// TIA Portal V17 export
// export: Created 2025-03-05T07:59:12.9568395Z, ExportSetting WithDefaults, DisplayName Totally Integrated Automation Portal, DisplayVersion V17 Update 8, DisplayName TIA Portal Openness, DisplayVersion V17 Update 8, DisplayName TIA Portal Version Control Interface, DisplayVersion V17, DisplayName SINAMICS Startdrive Advanced, DisplayVersion V17 SP2, DisplayName SINAMICS Startdrive G110M, G120, G120C, G120D, G120P, G115D, DisplayVersion V17 SP2, DisplayName SINAMICS Startdrive G130, G150, S120, S150, SINAMICS MV, S210, DisplayVersion V17 SP2, DisplayName STEP 7 Professional, DisplayVersion V17 Update 8, DisplayName SINUMERIK ONE STEP 7 Toolbox, DisplayVersion V17 Update 12, DisplayName SINUMERIK 840D sl STEP 7 Toolbox, DisplayVersion V17 Update 12, DisplayName STEP 7 Safety, DisplayVersion V17 Update 6, DisplayName WinCC Advanced, DisplayVersion V17 Update 8
DATA_BLOCK "DB4021_JAW_CHUCK_CONTROL_U02_STA_1"   // DB4021
{ S7_Optimized_Access := 'FALSE'; DB_Accessible_From_OPC_UA := 'FALSE' }
VERSION : 0.1
// stored: AutoNumber false, DBAccessibleFromOPCUA false, DBAccessibleFromWebserver true, IsOnlyStoredInLoadMemory false, IsWriteProtectedInAS false
   VAR RETAIN
      SENSOR_VALUE : UInt;   // UNIT 02 STATION 1 FIXTURE POSITION ANALOG VALUE
      UNCLAMPED_MAX : UInt;   // UNIT 02 STATION 1 FIXTURE UNCLAMPED MAX VALUE
      UNCLAMPED_MIN : UInt;   // UNIT 02 STATION 1 FIXTURE UNCLAMPED MIN VALUE
      CLAMPED_WITHOUT_PART_MAX : UInt;   // UNIT 02 STATION 1 FIXTURE CLAMPED NO PART MAX VALUE
      CLAMPED_WITHOUT_PART_MIN : UInt;   // UNIT 02 STATION 1 FIXTURE CLAMPED NO PART MIN VALUE
      CLAMPED_PART_1_MAX : UInt;   // UNIT 02 STATION 1 FIXTURE CLAMPED PART TYPE 1 MAX VALUE
      CLAMPED_PART_1_MIN : UInt;   // UNIT 02 STATION 1 FIXTURE CLAMPED PART TYPE 1 MIN VALUE
      CLAMPED_PART_2_MAX : UInt;   // UNIT 02 STATION 1 FIXTURE CLAMPED PART TYPE 2 MAX VALUE
      CLAMPED_PART_2_MIN : UInt;   // UNIT 02 STATION 1 FIXTURE CLAMPED PART TYPE 2 MAX VALUE
      CLAMPED_PART_3_MAX : UInt;   // UNIT 02 STATION 1 FIXTURE CLAMPED PART TYPE 3 MAX VALUE
      CLAMPED_PART_3_MIN : UInt;   // UNIT 02 STATION 1 FIXTURE CLAMPED PART TYPE 3 MAX VALUE
      CLAMPED_PART_4_MAX : UInt;   // UNIT 02 STATION 1 FIXTURE CLAMPED PART TYPE 4 MAX VALUE
      CLAMPED_PART_4_MIN : UInt;   // UNIT 02 STATION 1 FIXTURE CLAMPED PART TYPE 4 MAX VALUE
      CLAMPED_PART_5_MAX : UInt;   // UNIT 02 STATION 1 FIXTURE CLAMPED PART TYPE 5 MAX VALUE
      CLAMPED_PART_5_MIN : UInt;   // UNIT 02 STATION 1 FIXTURE CLAMPED PART TYPE 5 MAX VALUE
      CLAMPED_PART_6_MAX : UInt;   // UNIT 02 STATION 1 FIXTURE CLAMPED PART TYPE 6 MAX VALUE
      CLAMPED_PART_6_MIN : UInt;   // UNIT 02 STATION 1 FIXTURE CLAMPED PART TYPE 6 MAX VALUE
      CLAMPED_PART_7_MAX : UInt;   // UNIT 02 STATION 1 FIXTURE CLAMPED PART TYPE 7 MAX VALUE
      CLAMPED_PART_7_MIN : UInt;   // UNIT 02 STATION 1 FIXTURE CLAMPED PART TYPE 7 MAX VALUE
      CLAMPED_PART_8_MAX : UInt;   // UNIT 02 STATION 1 FIXTURE CLAMPED PART TYPE 8 MAX VALUE
      CLAMPED_PART_8_MIN : UInt;   // UNIT 02 STATION 1 FIXTURE CLAMPED PART TYPE 8 MAX VALUE
      CLAMPED_PART_9_MAX : UInt;   // UNIT 02 STATION 1 FIXTURE CLAMPED PART TYPE 9 MAX VALUE
      CLAMPED_PART_9_MIN : UInt;   // UNIT 02 STATION 1 FIXTURE CLAMPED PART TYPE 9 MAX VALUE
      CLAMPED_PART_10_MAX : UInt;   // UNIT 02 STATION 1 FIXTURE CLAMPED PART TYPE 10 MAX VALUE
      CLAMPED_PART_10_MIN : UInt;   // UNIT 02 STATION 1 FIXTURE CLAMPED PART TYPE 10 MAX VALUE
      CLAMPED_MASTER_MAX : UInt := 230;   // UNIT 02 STATION 1 FIXTURE CLAMPED WITH MASTER MAX VALUE
      CLAMPED_MASTER_MIN : UInt := 150;   // UNIT 02 STATION 1 FIXTURE CLAMPED WITH MASTER MIN VALUE
      SPARE_MIN_MAX : Array[1..39] of Real;
      UNCLAMPED : Bool;   // UNIT 02 STATION 1 FIXTURE UNCLAMPED
      CLAMPED_WITHOUT_PART : Bool;   // UNIT 02 STATION 1 FIXTURE CLAMPED WITH NO PART
      CLAMPED_PART_1 : Bool;   // UNIT 02 STATION 1 FIXTURE CLAMPED WITH PART TYPE 1
      CLAMPED_PART_2 : Bool;   // UNIT 02 STATION 1 FIXTURE CLAMPED WITH PART TYPE 2
      CLAMPED_PART_3 : Bool;   // UNIT 02 STATION 1 FIXTURE CLAMPED WITH PART TYPE 3
      CLAMPED_PART_4 : Bool;   // UNIT 02 STATION 1 FIXTURE CLAMPED WITH PART TYPE 4
      CLAMPED_PART_5 : Bool;   // UNIT 02 STATION 1 FIXTURE CLAMPED WITH PART TYPE 5
      CLAMPED_PART_6 : Bool;   // UNIT 02 STATION 1 FIXTURE CLAMPED WITH PART TYPE 6
      CLAMPED_PART_7 : Bool;   // UNIT 02 STATION 1 FIXTURE CLAMPED WITH PART TYPE 7
      CLAMPED_PART_8 : Bool;   // UNIT 02 STATION 1 FIXTURE CLAMPED WITH PART TYPE 8
      CLAMPED_PART_9 : Bool;   // UNIT 02 STATION 1 FIXTURE CLAMPED WITH PART TYPE 9
      CLAMPED_PART_10 : Bool;   // UNIT 02 STATION 1 FIXTURE CLAMPED WITH PART TYPE 10
      CLAMPED_MASTER : Bool := FALSE;   // UNIT 01 STATION 1 FIXTURE CLAMPED WITH MASTER
      SPARE_BOOL : Array[1..19] of Bool;
      CLAMPED_ANY_PART : Bool;   // UNIT 02 STATION 1 FIXTURE CLAMPED WITH ANY PART
      CLAMPED : Bool;   // UNIT 02 STATION 1 FIXTURE CLAMPED
   END_VAR
BEGIN
END_DATA_BLOCK
